// TIA Portal V16 export
// export: Created 2021-03-04T22:04:00.0558032Z, ExportSetting WithDefaults, DisplayName Totally Integrated Automation Portal, DisplayVersion V16, DisplayName TIA Portal Version Control Interface, DisplayVersion V16, DisplayName TIA Portal Openness, DisplayVersion V16, DisplayName SINAMICS Startdrive Advanced, DisplayVersion V16, DisplayName SINAMICS Startdrive G130, G150, S120, S150, SINAMICS MV, S210, DisplayVersion V16, DisplayName SINAMICS Startdrive G110M, G120, G120C, G120D, G120P, DisplayVersion V16, DisplayName STEP 7 Professional, DisplayVersion V16, DisplayName STEP 7 Safety, DisplayVersion V16, DisplayName WinCC Professional, DisplayVersion V16
FUNCTION_BLOCK "fbRoom"   // FB3, LAD
{ S7_Optimized_Access := 'TRUE' }
VERSION : 0.1
// stored: AutoNumber true, IsIECCheckEnabled false, IsRetainMemResEnabled false, MemoryReserve 100, SetENOAutomatically false, UDAEnableTagReadback false
   VAR_INPUT
      arrAI { ExternalAccessible := 'False'; ExternalVisible := 'False'; ExternalWritable := 'False'} : Array[1.."NUM_AI_ROOM"] of Int;
      AI AT arrAI : "udtRoomAI";
   END_VAR
   VAR_OUTPUT
      arrDQ { ExternalAccessible := 'False'; ExternalVisible := 'False'; ExternalWritable := 'False'} : Array[1.."NUM_DQ_ROOM"] of Bool;
      DQ AT arrDQ : "udtRoomDQ";
   END_VAR
   VAR
      Rack { ExternalVisible := 'False'} : Array[1.."MAX_RACKS_PER_ROOM"] of "fbRack";
      Fertigation { ExternalVisible := 'False'} : "fbRoomFertigation";
      HVAC { ExternalVisible := 'False'} : "fbRoomHVAC";
   END_VAR
   VAR RETAIN
      Config { ExternalVisible := 'False'; ExternalWritable := 'False'} : Struct
         iNumRacks { ExternalVisible := 'False'; ExternalWritable := 'False'} : Int := 1;
      END_STRUCT;
   END_VAR
   VAR
      AI_Temperature_1 { ExternalVisible := 'False'} : "fbAlarmedSetpoint";
      AI_Temperature_2 { ExternalVisible := 'False'} : "fbAlarmedSetpoint";
      AI_Humidity_1 { ExternalVisible := 'False'} : "fbAlarmedSetpoint";
      AI_Humidity_2 { ExternalVisible := 'False'} : "fbAlarmedSetpoint";
      AI_TankLevel { ExternalVisible := 'False'} : "fbAlarmedSetpoint";
      AI_NutrientALevel { ExternalVisible := 'False'} : "fbAlarmedSetpoint";
      AI_NutrientBLevel { ExternalVisible := 'False'} : "fbAlarmedSetpoint";
      AI_NutrientAcidLevel { ExternalVisible := 'False'} : "fbAlarmedSetpoint";
      AI_pHSensor { ExternalVisible := 'False'} : "fbAlarmedSetpoint";
      AI_ECSensor { ExternalVisible := 'False'} : "fbAlarmedSetpoint";
      AI_ISESensor { ExternalVisible := 'False'} : "fbAlarmedSetpoint";
      AI_ORPSensor { ExternalVisible := 'False'} : "fbAlarmedSetpoint";
   END_VAR
   VAR RETAIN
      DQ_MPathSolenoid { ExternalVisible := 'False'} : "udtDigitalOutput";
      DQ_FreshWaterSolenoid { ExternalVisible := 'False'} : "udtDigitalOutput";
      DQ_DischargeSolenoid { ExternalVisible := 'False'} : "udtDigitalOutput";
      DQ_TankReturnSolenoid { ExternalVisible := 'False'} : "udtDigitalOutput";
      DQ_NutrientA { ExternalVisible := 'False'} : "udtDigitalOutput";
      DQ_NutrientB { ExternalVisible := 'False'} : "udtDigitalOutput";
      DQ_NutrientAcid { ExternalVisible := 'False'} : "udtDigitalOutput";
      DQ_NutrientMixing { ExternalVisible := 'False'} : "udtDigitalOutput";
      DQ_CO2Solenoid { ExternalVisible := 'False'} : "udtDigitalOutput";
   END_VAR
   VAR
      arrFertigationSettings { ExternalAccessible := 'False'; ExternalVisible := 'False'; ExternalWritable := 'False'} : Array[0.."MAX_RACKS_PER_ROOM"] of "udtFertigationSettings";
   END_VAR
   VAR_TEMP
      i : Int;   // Index for iterating through racks
      max_temp : Int;
   END_VAR
   // AI_Temperature_1.Config.rLowCalibration := -40.0;
   // AI_Temperature_1.Config.rHighCalibration := 140.0;
   // AI_Temperature_2.Config.rLowCalibration := -40.0;
   // AI_Temperature_2.Config.rHighCalibration := 140.0;
   // AI_Humidity_1.Config.rLowCalibration := 0.0;
   // AI_Humidity_1.Config.rHighCalibration := 100.0;
   // AI_Humidity_2.Config.rLowCalibration := 0.0;
   // AI_Humidity_2.Config.rHighCalibration := 100.0;
   // AI_TankLevel.Config.rLowCalibration := 0.0;
   // AI_TankLevel.Config.rHighCalibration := 1085.0;
   // AI_NutrientALevel.Config.rLowCalibration := 0.0;
   // AI_NutrientALevel.Config.rHighCalibration := 200.0;
   // AI_NutrientBLevel.Config.rLowCalibration := 0.0;
   // AI_NutrientBLevel.Config.rHighCalibration := 200.0;
   // AI_NutrientAcidLevel.Config.rLowCalibration := 0.0;
   // AI_NutrientAcidLevel.Config.rHighCalibration := 200.0;
   // AI_pHSensor.Config.rLowCalibration := 0.0;
   // AI_pHSensor.Config.rHighCalibration := 14.0;
   // AI_ECSensor.Config.rLowCalibration := 0.0;
   // AI_ECSensor.Config.rHighCalibration := 5.0;
   // AI_ISESensor.Config.rLowCalibration := 0.0;
   // AI_ISESensor.Config.rHighCalibration := 10000.0;
   // AI_ORPSensor.Config.rLowCalibration := -1500.0;
   // AI_ORPSensor.Config.rHighCalibration := 1500.0;
BEGIN

REGION Network 1 (SCL): Process room-level analog inputs
   #AI_Temperature_1(#AI.IW_RoomTemperature_1);
   #AI_Temperature_2(#AI.IW_RoomTemperature_2);
   #AI_Humidity_1(#AI.IW_RoomHumidity_1);
   #AI_Humidity_2(#AI.IW_RoomHumidity_2);
   #AI_TankLevel(#AI.IW_TankLevel);
   #AI_NutrientALevel(#AI.IW_NutrientALevel);
   #AI_NutrientBLevel(#AI.IW_NutrientBLevel);
   #AI_NutrientAcidLevel(#AI.IW_NutrientAcidLevel);
   #AI_pHSensor(#AI.IW_pHSensor);
   #AI_ECSensor(#AI.IW_ECSensor);
   #AI_ISESensor(#AI.IW_ISESensor);
   #AI_ORPSensor(#AI.IW_ORPSensor);
   //#AI_CO2Sensor(#AI.IW_CO2Sensor);
END_REGION

REGION Network 2 (SCL): Call rack FBs
   #max_temp := MAX(IN1 := #AI_Temperature_1.rActual, IN2 := #AI_Temperature_2.rActual);
   #max_temp := MAX(IN1 := #max_temp, IN2 := #HVAC.Temperature_Cooling.rActual);

   FOR #i := 1 TO #Config.iNumRacks DO

       #Rack[#i](iInMutexLockConfirmation := #Fertigation.arrOutMutexLocks[#i],
                 udtInLastNutrientReading := #Fertigation.arrOutNutrientReading[#i],
                 bInSupplySolenoidFromRoomFertigation := #Fertigation.arrOutSupplySolenoids[#i],
                 bInReturnSolenoidFromRoomFertigation := #Fertigation.arrOutReturnSolenoids[#i],
                 iInLightsDelaySecs := #i * 5000, // delay each rack by 5 seconds to prevent current spike
                 arrAI := #Rack[#i].arrAI,
                 rInCurrentTemperature := #max_temp,
                 iOutMutexRequest => #Fertigation.arrInMutexRequests[#i],
                 OutFertigationSettings => #arrFertigationSettings[#i],
                 arrDQ => #Rack[#i].arrDQ);
   END_FOR;
END_REGION

REGION Network 3 (SCL): Call room-level fertigation control logic and map rack supply and return solenoids
   #Fertigation(arrInMutexRequests:=#Fertigation.arrInMutexRequests,
                arrInFertigationSettings:=#arrFertigationSettings,
                rInTankLevel:=#AI_TankLevel.rActual,
                rInNutrientALevel:=#AI_NutrientALevel.rActual,
                rInNutrientBLevel:=#AI_NutrientBLevel.rActual,
                rInNutrientAcidLevel:=#AI_NutrientAcidLevel.rActual,
                rInpHSensor:=#AI_pHSensor.rActual,
                rInECSensor:=#AI_ECSensor.rActual,
                rInISESensor:=#AI_ISESensor.rActual,
                rInORPReading:=#AI_ORPSensor.rActual,
                iInNumRacks:=#Config.iNumRacks,
                bOutTankReturnSolenoid=>#Fertigation.bOutTankReturnSolenoid,
                bOutMPathSolenoid=>#Fertigation.bOutMPathSolenoid,
                bOutFreshWaterSolenoid=>#Fertigation.bOutFreshWaterSolenoid,
                bOutDischargeSolenoid=>#Fertigation.bOutDischargeSolenoid,
                bOutNutrientMixing=>#Fertigation.bOutNutrientMixing,
                bOutNutrientA=>#Fertigation.bOutNutrientA,
                bOutNutrientB=>#Fertigation.bOutNutrientB,
                bOutNutrientAcid=>#Fertigation.bOutNutrientAcid,
                arrOutNutrientReading=>#Fertigation.arrOutNutrientReading,
                arrOutMutexLocks=>#Fertigation.arrOutMutexLocks,
                arrOutSupplySolenoids=>#Fertigation.arrOutSupplySolenoids,
                arrOutReturnSolenoids=>#Fertigation.arrOutReturnSolenoids);
END_REGION

REGION Network 4 (SCL): Call HVAC and CO2 control logic
   #HVAC(iInCO2ReadingRaw := #AI.IW_CO2Sensor,
         bOutCO2Solenoid=>#HVAC.bOutCO2Solenoid);
END_REGION

REGION Network 5 (SCL): Set room-level outputs
   #DQ.Q_MPathSolenoid := "fcDigitalOutput"(bInAutoVal := #Fertigation.bOutMPathSolenoid, InOutUdt := #DQ_MPathSolenoid);
   #DQ.Q_FreshWaterSolenoid := "fcDigitalOutput"(bInAutoVal := #Fertigation.bOutFreshWaterSolenoid, InOutUdt := #DQ_FreshWaterSolenoid);
   #DQ.Q_DischargeSolenoid := "fcDigitalOutput"(bInAutoVal := #Fertigation.bOutDischargeSolenoid, InOutUdt := #DQ_DischargeSolenoid);
   #DQ.Q_TankReturnSolenoid := "fcDigitalOutput"(bInAutoVal := #Fertigation.bOutTankReturnSolenoid, InOutUdt := #DQ_TankReturnSolenoid);
   #DQ.Q_NutrientAEnable := "fcDigitalOutput"(bInAutoVal := #Fertigation.bOutNutrientA, InOutUdt := #DQ_NutrientA);
   #DQ.Q_NutrientBEnable := "fcDigitalOutput"(bInAutoVal := #Fertigation.bOutNutrientB, InOutUdt := #DQ_NutrientB);
   #DQ.Q_NutrientAcidEnable := "fcDigitalOutput"(bInAutoVal := #Fertigation.bOutNutrientAcid, InOutUdt := #DQ_NutrientAcid);
   #DQ.Q_NutrientMixingPumps := "fcDigitalOutput"(bInAutoVal := #Fertigation.bOutNutrientMixing, InOutUdt := #DQ_NutrientMixing);

   #DQ.Q_CO2Solenoid := "fcDigitalOutput"(bInAutoVal := #HVAC.bOutCO2Solenoid, InOutUdt := #DQ_CO2Solenoid);
END_REGION
END_FUNCTION_BLOCK
